// TwinCAT 3 PLC project SPS
// ProgramVersion: 3.1.4024.0
// libraries:
//   Tc2_MC2, * (Beckhoff Automation GmbH)
//   Tc2_Standard, * (Beckhoff Automation GmbH)
//   Tc2_System, * (Beckhoff Automation GmbH)
//   Tc3_IotBase, * (Beckhoff Automation GmbH)
//   Tc3_Module, * (Beckhoff Automation GmbH)
// project tree:
//   DUTs/ eBetriebszustand.TcDUT
//   GVLs/ GVL_PosKinematic.TcGVL, IFC_HW.TcGVL (not stored)
//   / PlcTask.TcTTO
//   POUs/ FB_Abfullmodul.TcPOU, FB_Ampel.TcPOU, FB_Blinklicht.TcPOU, FB_Dispenser.TcPOU, FB_EZylinder.TcPOU, FB_IotMqttCommunication.TcPOU, FB_ManipulatorAchsen.TcPOU, FB_Vereinzelung.TcPOU, FUN_Scale.TcPOU, MAIN.TcPOU
//   POUs/PortalRoboter/ FB_AchsenRoboter.TcPOU, FB_Robotersteuerung.TcPOU, FB_Thermo_Temp.TcPOU, FB_Waage_Temp.TcPOU
//   POUs/Transport/ FB_TransportBand.TcPOU, FB_Transport.TcPOU, FB_TransportA.TcPOU, FB_TransportLogik.TcPOU, FB_TransportE.TcPOU
// real-time tasks:
//   TASK PlcTask: cycle T#10ms, priority 20, ADS port 350
//   TASK PlcTask1: cycle T#10ms, priority 21, ADS port 351
// motion (NC):
//   TASK NC-Task 1 SAF: cycle T#2ms, priority 4, ADS port 501
//   TASK NC-Task 1 SVB: cycle T#10ms, priority 8, ADS port 511
//   AXIS Achse_ManG (id 7)
//     OtherSettings: AllowMotionCmdToSlave=true
//     encoder EncType=1
//       EncPara: ScaleFactorNumerator=0.0025
//         Inc: RefSearchInverse=true, RefSyncInverse=false
//     drive DrvType=5
//       Analog: TorqueSetpointScale=10, ScaleFactorActTorque=0.1
//       TimeComp: TaskDelayCycles=1
//     controller CtrType=1
//       CtrPara: PriorControlFactor=1
//         Observer: BandWidth=20
//   AXIS Achse_Band (id 1)
//     OtherSettings: AllowMotionCmdToSlave=true
//     encoder EncType=1
//     drive DrvType=5
//       Analog: TorqueSetpointScale=10, ScaleFactorActTorque=0.1
//       TimeComp: TaskDelayCycles=1
//     controller CtrType=1
//       CtrPara: PriorControlFactor=1
//         Observer: BandWidth=20
//   AXIS Achse_Dispenser1 (id 2)
//     OtherSettings: AllowMotionCmdToSlave=true
//     encoder EncType=1
//     drive DrvType=5
//       Analog: TorqueSetpointScale=10, ScaleFactorActTorque=0.1
//       TimeComp: TaskDelayCycles=1
//     controller CtrType=1
//       CtrPara: PriorControlFactor=1
//         Observer: BandWidth=20
//   AXIS Achse_Dispenser2 (id 3)
//     OtherSettings: AllowMotionCmdToSlave=true
//     encoder EncType=1
//     drive DrvType=5
//       Analog: TorqueSetpointScale=10, ScaleFactorActTorque=0.1
//       TimeComp: TaskDelayCycles=1
//     controller CtrType=1
//       CtrPara: PriorControlFactor=1
//         Observer: BandWidth=20
//   AXIS Achse_Dispenser3 (id 4)
//     OtherSettings: AllowMotionCmdToSlave=true
//     encoder EncType=1
//     drive DrvType=5
//       Analog: TorqueSetpointScale=10, ScaleFactorActTorque=0.1
//       TimeComp: TaskDelayCycles=1
//     controller CtrType=1
//       CtrPara: PriorControlFactor=1
//         Observer: BandWidth=20
//   AXIS Achse_ManX (id 5)
//     OtherSettings: AllowMotionCmdToSlave=true
//     encoder EncType=1
//       EncPara: ScaleFactorNumerator=0.0025
//         Inc: RefSearchInverse=true, RefSyncInverse=false
//     drive DrvType=5
//       Analog: TorqueSetpointScale=10, ScaleFactorActTorque=0.1
//       TimeComp: TaskDelayCycles=1
//     controller CtrType=1
//       CtrPara: PriorControlFactor=1
//         Observer: BandWidth=20
//   AXIS Achse_ManY (id 6)
//     OtherSettings: AllowMotionCmdToSlave=true
//     encoder EncType=1
//       EncPara: ScaleFactorNumerator=0.0025
//         Inc: RefSearchInverse=true, RefSyncInverse=false
//     drive DrvType=5
//       Analog: TorqueSetpointScale=10, ScaleFactorActTorque=0.1
//       TimeComp: TaskDelayCycles=1
//     controller CtrType=1
//       CtrPara: PriorControlFactor=1
//         Observer: BandWidth=20
//   AXIS Achse_ManZ (id 8)
//     OtherSettings: AllowMotionCmdToSlave=true
//     encoder EncType=1
//       EncPara: ScaleFactorNumerator=0.0025
//         Inc: RefSearchInverse=true, RefSyncInverse=false
//     drive DrvType=5
//       Analog: TorqueSetpointScale=10, ScaleFactorActTorque=0.1
//       TimeComp: TaskDelayCycles=1
//     controller CtrType=1
//       CtrPara: PriorControlFactor=1
//         Observer: BandWidth=20
// I/O:
//   DEVICE Gerät 3 (EtherCAT) (disabled), AmsNetId 192.168.137.1.4.1
//     Klemme 1 (EK1100) [EK1100 EtherCAT-Koppler (2A E-Bus)]
//       Klemme 2 (EL1014) [EL1014 4K. Dig. Eingang 24V, 10µs]
//       Klemme 3 (EL2008) [EL2008 8K. Dig. Ausgang 24V, 0.5A]
//       Klemme 4 (EL2008) [EL2008 8K. Dig. Ausgang 24V, 0.5A]
//       Klemme 5 (EL9011) [EL9011 Endklemme]
// variable links:
//   SPS/SPS Instance <-> Device 3 (EtherCAT)/Term 1 (EK1100)/Term 2 (EL1014)
//     PlcTask Inputs/IFC_HW.bExecute <-> Channel 1/Input
//   SPS/SPS Instance <-> Device 3 (EtherCAT)/Term 1 (EK1100)/Term 3 (EL2008)
//     PlcTask Outputs/IFC_HW.bAmpelRot <-> Channel 1/Output
//   SPS/SPS Instance <-> NC-Task 1 SAF/Axes/Achse_Band
//     PlcTask Inputs/IFC_HW.ax_BandMotor.NcToPlc <-> Outputs/ToPlc
//     PlcTask Outputs/IFC_HW.ax_BandMotor.PlcToNc <-> Inputs/FromPlc
//   SPS/SPS Instance <-> NC-Task 1 SAF/Axes/Achse_Dispenser1
//     PlcTask Inputs/IFC_HW.ax_Extruder1.NcToPlc <-> Outputs/ToPlc
//     PlcTask Outputs/IFC_HW.ax_Extruder1.PlcToNc <-> Inputs/FromPlc
//   SPS/SPS Instance <-> NC-Task 1 SAF/Axes/Achse_Dispenser2
//     PlcTask Inputs/IFC_HW.ax_Extruder2.NcToPlc <-> Outputs/ToPlc
//     PlcTask Outputs/IFC_HW.ax_Extruder2.PlcToNc <-> Inputs/FromPlc
//   SPS/SPS Instance <-> NC-Task 1 SAF/Axes/Achse_Dispenser3
//     PlcTask Inputs/IFC_HW.ax_Extruder3.NcToPlc <-> Outputs/ToPlc
//     PlcTask Outputs/IFC_HW.ax_Extruder3.PlcToNc <-> Inputs/FromPlc
//   SPS/SPS Instance <-> NC-Task 1 SAF/Axes/Achse_ManG
//     PlcTask Inputs/IFC_HW.ax_ManG.NcToPlc <-> Outputs/ToPlc
//     PlcTask Outputs/IFC_HW.ax_ManG.PlcToNc <-> Inputs/FromPlc
//   SPS/SPS Instance <-> NC-Task 1 SAF/Axes/Achse_ManX
//     PlcTask Inputs/IFC_HW.ax_ManX.NcToPlc <-> Outputs/ToPlc
//     PlcTask Outputs/IFC_HW.ax_ManX.PlcToNc <-> Inputs/FromPlc
//   SPS/SPS Instance <-> NC-Task 1 SAF/Axes/Achse_ManY
//     PlcTask Inputs/IFC_HW.ax_ManY.NcToPlc <-> Outputs/ToPlc
//     PlcTask Outputs/IFC_HW.ax_ManY.PlcToNc <-> Inputs/FromPlc
//   SPS/SPS Instance <-> NC-Task 1 SAF/Axes/Achse_ManZ
//     PlcTask Inputs/IFC_HW.ax_ManZ.NcToPlc <-> Outputs/ToPlc
//     PlcTask Outputs/IFC_HW.ax_ManZ.PlcToNc <-> Inputs/FromPlc

CONFIGURATION SPS
    RESOURCE PLC ON TwinCAT3
        TASK PlcTask(INTERVAL := T#10ms, PRIORITY := 20);
        PROGRAM MAIN WITH PlcTask : MAIN;
    END_RESOURCE
END_CONFIGURATION

// ---- DUTs/eBetriebszustand.TcDUT
{attribute 'qualified_only'}
{attribute 'strict'}
TYPE eBetriebszustand :
(
	Off , //Nicht Betriebsbereit, ROT
	Error , //Fehlerbehafteter Stop (Sicherheitssteuerung), ROT blinkend
	Setup , //Wartung, GELB
	Warning , //Nicht Fehlerbehafteter aber nicht geplanter Stop, GELB blinkend
	Init ,  //herstellung Betriebsbereitschaft, GELB GRÜN
	Ready , // Betriebsbereitschaft, GRÜN
	Production , //Betrieb, GRÜN GELB blinkend
	Done, //Betrieb abgeschlossen, GRÜN blinkend
	Stop //Geplanter Stopp ROT GELB blinkend
	
);
END_TYPE

// ---- GVLs/GVL_PosKinematic.TcGVL
{attribute 'qualified_only'}
VAR_GLOBAL
	// Home position
	pXhome : REAL := 29;
	pYhome : REAL := 145.5;
	pZhome : REAL := 45;
	
	// Conveyor position
	pXconv : REAL := 29;
	pYconv : REAL := 145.5;
	pZconv : REAL := 130;
	
	//Scale position
	pXscale : REAL := 36;
	pYscale : REAL := 7.5;
	pZscale : REAL := 131.5;
	
	// Heating position
	pXheat : REAL := 218.5;
	pYheat : REAL := 7;
	pZheat : REAL := 159;
	
	// Storage position
	pX1stor : REAL := 107;
	pX2stor : REAL := 158.7;
	pX3stor : REAL := 209.3;
	pX4stor : REAL := 260.3;
	pYstor : REAL := 139;
	pZstor : REAL := 120;
	
	// Z offset height
	pZoff : REAL := 45;
END_VAR

// ---- POUs/MAIN.TcPOU
PROGRAM MAIN
VAR
	fbAmpel : FB_Ampel;
	fbEZylinder1 : FB_EZylinder;
	fbEZylinder2 : FB_EZylinder;
	MCPowerBand : MC_Power;
	MCPowerDispenser1 	: MC_Power;
	MCPowerDispenser2 	: MC_Power;
	MCPowerDispenser3 	: MC_Power;
	MCPowerAchseX	 	: MC_Power;
	MCPowerAchseY 	: MC_Power;
	MCPowerAchseZ 	: MC_Power;
	MCPowerAchseG 	: MC_Power;
	fbAbfullModul : FB_Abfullmodul;
	fbRoboter : FB_Robotersteuerung;
	fbIotMqttCommunication : FB_IotMqttCommunication;
	
	nRoboterLagerIndex : INT;
	

	ix : REAL;
	ry : UINT;
	
	
  	

END_VAR

ry := TO_UINT(FUN_Scale(ix,4096, 0, 350, 0));

IFC_HW.ax_BandMotor.ReadStatus();
IFC_HW.ax_Extruder1.ReadStatus();
IFC_HW.ax_Extruder2.ReadStatus();
IFC_HW.ax_Extruder3.ReadStatus();



MCPowerBand(
	Axis:= IFC_HW.ax_BandMotor , 
	Enable:= TRUE , 
	Enable_Positive:= TRUE, 
	Enable_Negative:= TRUE, 
	Override:= , 
	BufferMode:= , 
	Options:= , 
	Status=> , 
	Busy=> , 
	Error=> , 
	ErrorID=> );
	
MCPowerDispenser1(
	Axis:= IFC_HW.ax_Extruder1, 
	Enable:= TRUE, 
	Enable_Positive:= TRUE, 
	Enable_Negative:= TRUE, 
	Override:= , 
	BufferMode:= , 
	Options:= , 
	Status=> , 
	Busy=> , 
	Error=> , 
	ErrorID=> );
	
MCPowerDispenser2(
	Axis:= IFC_HW.ax_Extruder2, 
	Enable:= TRUE, 
	Enable_Positive:= TRUE, 
	Enable_Negative:= TRUE, 
	Override:= , 
	BufferMode:= , 
	Options:= , 
	Status=> , 
	Busy=> , 
	Error=> , 
	ErrorID=> );
	
MCPowerDispenser3(
	Axis:= IFC_HW.ax_Extruder3, 
	Enable:= TRUE, 
	Enable_Positive:= TRUE, 
	Enable_Negative:= TRUE, 
	Override:= , 
	BufferMode:= , 
	Options:= , 
	Status=> , 
	Busy=> , 
	Error=> , 
	ErrorID=> );
	
MCPowerAchseX(
	Axis:= IFC_HW.ax_ManX, 
	Enable:= TRUE, 
	Enable_Positive:= TRUE, 
	Enable_Negative:= TRUE, 
	Override:= , 
	BufferMode:= , 
	Options:= , 
	Status=> , 
	Busy=> , 
	Error=> , 
	ErrorID=> );
	
MCPowerAchseY(
	Axis:= IFC_HW.ax_ManY, 
	Enable:= TRUE, 
	Enable_Positive:= TRUE, 
	Enable_Negative:= TRUE, 
	Override:= , 
	BufferMode:= , 
	Options:= , 
	Status=> , 
	Busy=> , 
	Error=> , 
	ErrorID=> );

MCPowerAchseZ(
	Axis:= IFC_HW.ax_ManZ, 
	Enable:= TRUE, 
	Enable_Positive:= TRUE, 
	Enable_Negative:= TRUE, 
	Override:= , 
	BufferMode:= , 
	Options:= , 
	Status=> , 
	Busy=> , 
	Error=> , 
	ErrorID=> );
	
MCPowerAchseG(
	Axis:= IFC_HW.ax_ManG, 
	Enable:= TRUE, 
	Enable_Positive:= TRUE, 
	Enable_Negative:= TRUE, 
	Override:= , 
	BufferMode:= , 
	Options:= , 
	Status=> , 
	Busy=> , 
	Error=> , 
	ErrorID=> );


fbAbfullModul(
	bEnable:= IFC_HW.bEnable, 
	bExecute:= IFC_HW.bExecute, 
	bBandSens1:= IFC_HW.bBandSens1, 
	bBandSens2:= IFC_HW.bBandSens2, 
	bBandSens3:= IFC_HW.bBandSens3, 
	bBandSens4:= IFC_HW.bBandSens4, 
	bEinzelSens1:= IFC_HW.bEinzelSens1 , 
	bEinzelSens2:= IFC_HW.bEinzelSens2, 
	bEinzelSens3:= IFC_HW.bEinzelSens3, 
	nLagerIndex:= , 
	bGate1=> fbEZylinder1.bGate, 
	bGate2=> fbEZylinder2.bGate, 
	bStopper1=> IFC_HW.bBandHub1 , 
	bStopper2=> IFC_HW.bBandHub2, 
	bStopper3=> IFC_HW.bBandHub3, 
	eState=> , 
	axFoerderband:= IFC_HW.ax_BandMotor, 
	axDispenser1:= IFC_HW.ax_Extruder1, 
	axDispenser2:= IFC_HW.ax_Extruder2, 
	axDispenser3:= IFC_HW.ax_Extruder3
 );
 
 fbRoboter(
    bEnable := IFC_HW.bEnable,
    bExecute := IFC_HW.bExecute,

    bSensBand4 := IFC_HW.bBandSens4,
    bSensEndX := IFC_HW.bManEndXmin,
    bSensEndY := IFC_HW.bManEndYmin,
    bSensEndZ := IFC_HW.bManEndZmin,
    bSensEndG := IFC_HW.bManEndGmin,

    eState => ,

    bBrakeZ => IFC_HW.bManBrakeZ,
    bGripperClosed => IFC_HW.bGripperClosed,

    axX := IFC_HW.ax_ManX,
    axY := IFC_HW.ax_ManY,
    axZ := IFC_HW.ax_ManZ,
    axG := IFC_HW.ax_ManG,

    nLagerIndex := nRoboterLagerIndex
);
 
 fbIotMqttCommunication(
	sTopicToPublish:= 'bEnable',
	sMessageToPublish:= BOOL_TO_STRING(IFC_HW.bEnable),
);
	
fbEZylinder1(bGate:= , bError:= ,
			 bR1=> IFC_HW.bR1AKT1, bR2=> IFC_HW.bR2AKT1);
fbEZylinder2(bGate:= , bError:= , 
			bR1=> IFC_HW.bR1AKT2, bR2=> IFC_HW.bR2AKT2 );
			
fbAmpel(eState:= fbAbfullmodul.eState, bAmpelGrun=> IFC_HW.bAmpelGrun, bAmpelRot=> IFC_HW.bAmpelRot , bAmpelGelb=> IFC_HW.bAmpelGelb);

END_PROGRAM

// ---- POUs/FB_Ampel.TcPOU
FUNCTION_BLOCK FB_Ampel
VAR_INPUT
	eState : eBetriebszustand;
END_VAR
VAR_OUTPUT
	bAmpelGrun : BOOL;
	bAmpelRot : BOOL;
	bAmpelGelb : BOOL;
END_VAR
VAR
	fbBlinklicht : FB_Blinklicht;
END_VAR

CASE eState OF
	eBetriebszustand.Off:
		bAmpelGrun := FALSE;
		bAmpelGelb := FALSE;
		bAmpelRot := TRUE;
	
	eBetriebszustand.Error:
		bAmpelGrun := FALSE;
		bAmpelGelb := FALSE;
		fbBlinklicht(bStartStop:= TRUE, tPeriode:= T#1S, bBlink=> bAmpelRot );
	
	eBetriebszustand.Setup:
		bAmpelGrun := FALSE;
		bAmpelGelb := TRUE;
		bAmpelRot := FALSE;
	
	eBetriebszustand.Warning:
		bAmpelGrun := FALSE;
		fbBlinklicht(bStartStop:= TRUE, tPeriode:= T#1S, bBlink=> bAmpelGelb );
		bAmpelRot := FALSE;
		
	eBetriebszustand.Init:
		bAmpelGrun := TRUE;
		bAmpelGelb := TRUE;
		bAmpelRot := FALSE;
	
	eBetriebszustand.Ready:
		bAmpelGrun := TRUE;
		bAmpelGelb := FALSE;
		bAmpelRot := FALSE;
	
	eBetriebszustand.Production:
		bAmpelRot := FALSE;
		fbBlinklicht(bStartStop:= TRUE , tPeriode:= T#1S, bBlink=> bAmpelGrun);
		fbBlinklicht(bStartStop:= TRUE , tPeriode:= T#1S, bBlink=> bAmpelGelb);
	
	eBetriebszustand.Done:
		fbBlinklicht(bStartStop:= TRUE , tPeriode:= T#1S, bBlink=> bAmpelGrun);
		bAmpelGelb := FALSE;
		bAmpelRot := FALSE;
		
	eBetriebszustand.Stop:
		bAmpelGrun := FALSE;
		fbBlinklicht(bStartStop:= TRUE , tPeriode:= T#1S, bBlink=> bAmpelRot);
		fbBlinklicht(bStartStop:= TRUE , tPeriode:= T#1S, bBlink=> bAmpelGelb);
	
	
	
	
	
	
	
END_CASE

END_FUNCTION_BLOCK

// ---- POUs/FB_Blinklicht.TcPOU
FUNCTION_BLOCK FB_Blinklicht
VAR_INPUT
	bStartStop : BOOL;
	tPeriode : TIME := T#1S;
END_VAR
VAR_OUTPUT
	bBlink : BOOL;
END_VAR
VAR
	fbTon : Ton;
	fbRtrig : R_Trig;
	bEinAus : BOOL;
END_VAR


fbRtrig(CLK:= bStartStop, Q=>);
IF fbRtrig.Q THEN
	bEinAus := NOT bEinAus;
END_IF


//fbTon.IN := bBlink AND NOT fbTon.Q;
//fbTon.PT := T#1S;

fbTon(IN:= bEinAus AND NOT fbTon.Q , PT:= tPeriode , Q=>  , ET=> );

IF fbTon.ET <= fbTon.PT/2 THEN
	bBlink := FALSE;
ELSIF fbTon.ET > fbTon.PT/2 THEN
	bBlink := TRUE;
END_IF

END_FUNCTION_BLOCK

// ---- POUs/FB_EZylinder.TcPOU
FUNCTION_BLOCK FB_EZylinder
VAR_INPUT
	bGate : BOOL;
	bError : BOOL;
END_VAR
VAR_OUTPUT
	bR1 : BOOL;
	bR2 : BOOL;
END_VAR
VAR
END_VAR


bR1 := bGate;
bR2 := NOT bGate;

IF bError THEN
	bR1 := FALSE;
	bR2 := FALSE;
END_IF

END_FUNCTION_BLOCK

// ---- POUs/FB_Abfullmodul.TcPOU
FUNCTION_BLOCK FB_AbfullModul
VAR_INPUT
    bEnable     : BOOL;
    bExecute    : BOOL; 
	bBandSens1 	: BOOL;   
    bBandSens2 	: BOOL; 
	bBandSens3 	: BOOL; 
	bBandSens4 	: BOOL; 
 	bEinzelSens1: BOOL;
	bEinzelSens2: BOOL;
	bEinzelSens3: BOOL;
	nLagerIndex : INT;
END_VAR

VAR_OUTPUT
	//Vereinzelungsoutputs
	bGate1 : BOOL;
    bGate2 : BOOL;
	//Transportoutputs
	bStopper1 : BOOL;
    bStopper2 : BOOL;
    bStopper3 : BOOL;
    eState      : eBetriebszustand;
END_VAR

VAR
    fbVereinzelung      : FB_Vereinzelung;
    fbDispenser1         : FB_Dispenser;
	fbDispenser2         : FB_Dispenser;
	fbDispenser3         : FB_Dispenser;
    fbTransport    		: FB_Transport;
	
	fTrigBandSens4 : f_TRIG; 
	bBandSens4Rise  : BOOL;
	
    nState : INT := 0;
	nStation : INT;
	
	
END_VAR

VAR_IN_OUT
    axFoerderband : Axis_Ref;
    axDispenser1    : Axis_Ref;
	axDispenser2    : Axis_Ref;
	axDispenser3    : Axis_Ref;
   // axManipulator : Axis_Ref;
END_VAR

fbVereinzelung(
	bEnable:= bEnable, 
	bExecute:=  , 
	bSensor1:= bEinzelSens1, 
	bSensor2:= bEinzelSens2 , 
	bSensor3:= bEinzelSens3 , 
	bSensor4:= bBandSens1 , 
	bGate1=> bGate1 , 
	bGate2=> bGate2, 
	eState=> );
	
fbTransport(
	bEnable:= bEnable, 
	bExecute:= , 
	nStation:= nStation, 
	bSens1:= bBandSens1, 
	bSens2:= bBandSens2, 
	bSens3:= bBandSens3 , 
	bSens4:= bBandSens4, 
	eState=> , 
	bStopper1=> bStopper1, 
	bStopper2=> bStopper2, 
	bStopper3=> bStopper3, 
	ax:= axFoerderband);
	
fbDispenser1(
	bEnable:= bEnable, 
	bExecute:=, 
	rDistance:= , 
	eState=> , 
	ax:= axDispenser1);
	
fbDispenser2(
	bEnable:= bEnable, 
	bExecute:=, 
	rDistance:= , 
	eState=> , 
	ax:= axDispenser2);
	
fbDispenser3(
	bEnable:= bEnable, 
	bExecute:= , 
	rDistance:= , 
	eState=> , 
	ax:= axDispenser3);
	
	
CASE nState OF
	0: // OFF
	eState := eBetriebszustand.Off;
	fbVereinzelung.bEnable := FALSE;
	fbVereinzelung.bExecute := FALSE;
	fbTransport.bEnable := FALSE;
	fbTransport.bExecute := FALSE;
	fbDispenser1.bEnable := FALSE;
	fbDispenser2.bEnable := FALSE;
	fbDispenser3.bEnable := FALSE;
	fbDispenser1.bExecute := FALSE;
	fbDispenser2.bExecute := FALSE;
	fbDispenser3.bExecute := FALSE;
	
	
	IF bEnable THEN
		nState := 10;
	END_IF
	
	10: // INIT
	
	eState := eBetriebszustand.Init;
	fbVereinzelung.bEnable := TRUE;
	fbVereinzelung.bExecute := FALSE;
	fbTransport.bEnable := TRUE;
	fbTransport.bExecute := FALSE;
	fbDispenser1.bEnable := TRUE;
	fbDispenser2.bEnable := TRUE;
	fbDispenser3.bEnable := TRUE;
	fbDispenser1.bExecute := FALSE;
	fbDispenser2.bExecute := FALSE;
	fbDispenser3.bExecute := FALSE;
	
	IF fbVereinzelung.eState = eBetriebszustand.Ready AND fbTransport.eState = eBetriebszustand.Ready AND fbDispenser1.eState = eBetriebszustand.Ready AND fbDispenser2.eState = eBetriebszustand.Ready AND fbDispenser3.eState = eBetriebszustand.Ready THEN
		nState := 20;
	END_IF
	
	20: // READY
	eState := eBetriebszustand.Ready;
	fbVereinzelung.bEnable := TRUE;
	fbVereinzelung.bExecute := FALSE;
	fbTransport.bEnable := TRUE;
	fbTransport.bExecute := FALSE;
	fbDispenser1.bEnable := TRUE;
	fbDispenser2.bEnable := TRUE;
	fbDispenser3.bEnable := TRUE;
	fbDispenser1.bExecute := FALSE;
	fbDispenser2.bExecute := FALSE;
	fbDispenser3.bExecute := FALSE;
	
	IF bExecute THEN
		nState := 30;
	END_IF
	
	30: //Production
	eState := eBetriebszustand.Production;
	fbVereinzelung.bExecute := TRUE;
	fbTransport.bExecute := TRUE;
	fbDispenser1.bExecute := FALSE;
	fbDispenser2.bExecute := FALSE;
	fbDispenser3.bExecute := FALSE;
	nStation := 1;
	
	IF fbVereinzelung.eState = eBetriebszustand.Done AND fbTransport.eState = eBetriebszustand.Done THEN
		nState := 31;
	END_IF
	
	31: // 1st Dispenser
	nStation := 1;
	fbDispenser1.bExecute := TRUE;
	fbVereinzelung.bExecute := FALSE;
	fbTransport.bExecute := FALSE;
	
	IF fbDispenser1.eState = eBetriebszustand.Done THEN
		nState := 32;
	END_IF
	
	32: // Bewegung zu Station 2
	nStation := 2;
	fbTransport.bExecute := TRUE;
	fbDispenser1.bExecute := FALSE;
	
	IF fbTransport.eState = eBetriebszustand.Done THEN
		nState := 33;
	END_IF
	
	33: // 2nd Dispenser
	
	fbDispenser2.bExecute := TRUE;
	fbTransport.bExecute := FALSE;
	
	IF fbDispenser2.eState = eBetriebszustand.Done THEN
		nState := 34;
	END_IF
	
	34: //Bewegung zu Station 3
	nStation := 3;
	fbTransport.bExecute := TRUE;
	fbDispenser2.bExecute := FALSE;
	
	IF fbTransport.eState = eBetriebszustand.Done THEN
		nState := 35;
	END_IF
	
	35: //3rd Dispenser
	fbTransport.bExecute := FALSE;
	fbDispenser3.bExecute := TRUE;
	
	IF fbDispenser3.eState = eBetriebszustand.Done THEN
		nState := 36;
	END_IF
	
	36: // Bewegung zu Abholstation
	nStation := 4;
	fbDispenser3.bExecute := FALSE;
	fbTransport.bExecute := TRUE;
	
	IF fbTransport.eState = eBetriebszustand.Done THEN
		nState := 40;
	END_IF
	
	40: //DONE
	eState := eBetriebszustand.Done;
	fbTransport.bExecute := FALSE;
	
	
	IF NOT bExecute THEN
		nState := 20;
	END_IF
	
	
END_CASE

END_FUNCTION_BLOCK

// ---- POUs/FB_Vereinzelung.TcPOU
FUNCTION_BLOCK FB_Vereinzelung
VAR_INPUT
	//Steuervariablen
	bEnable : BOOL;
	bExecute : BOOL;
	//Hardware Eingänge
	bSensor1 : BOOL; // Flasche in der Kammer
	bSensor2 : BOOL; //Flasche im Rohr
	bSensor3 : BOOL; //Flasche auf Kopf
	bSensor4 : BOOL; //Flasche am Förderband
END_VAR
VAR_OUTPUT
	//Hardware Ausgänge
	bGate1 : BOOL;
	bGate2 : BOOL;
	//Steuervariable
	eState : eBetriebszustand;
END_VAR
VAR
	nState : INT := 100;
	fbTon : Ton;
END_VAR

fbTon(IN :=, PT := T#1S, Q=>, ET=>);
CASE nState OF
	100:
	eState := eBetriebszustand.Off;
	
	IF bSensor1 AND bEnable THEN
		nState := 21; //Ready
		ELSIF bEnable THEN
			nState := 0; //Init
	END_IF
	
	0: //Kammer ist Leer
	eState := eBetriebszustand.Init;
	bGate1 := FALSE;
	bGate2 := FALSE;
	
	IF bSensor2 THEN
		nState := 1; //Oben öffnen
	END_IF
	
	1: //Oben öffnen
	eState := eBetriebszustand.Init;
	bGate1 := TRUE;
	bGate2 := FALSE;
	
	IF bSensor1 THEN
		nState := 2; //oben schließen
	END_IF
	
	2: //oben Schließen
	eState := eBetriebszustand.Init;
	bGate1 := FALSE;
	bGate2 := FALSE;
	fbTon.IN := TRUE;
	
	
	IF fbTon.Q THEN
		nState := 21; //Ready
		fbTon.IN := FALSE;

	END_IF
	21: //Ready
	eState := eBetriebszustand.Ready;
	bGate1 := FALSE;
	bGate2 := FALSE;
	
	IF bExecute THEN
		nState := 3;
	END_IF
	
	3:
	eState := eBetriebszustand.Production;
	bGate1 := FALSE;
	bGate2 := TRUE;
	
	IF bSensor4 THEN
		nState := 4;
	END_IF
	
	4:
	eState := eBetriebszustand.Production;
	bGate1 := FALSE;
	bGate2 := FALSE;
	fbTon.IN := TRUE;
	
	IF fbTon.Q THEN
		nState := 41;
		fbTon.IN := FALSE;
		
	END_IF
	
	41: 
	eState := eBetriebszustand.Done;
	
	IF NOT bExecute THEN
		nState := 0;
		
	END_IF
	
	IF NOT bSensor2 AND bSensor3 THEN
		nState := 33;
	END_IF
	
	33:
	eState := eBetriebszustand.Warning;
	
	bExecute := FALSE;
	
	

	
END_CASE

END_FUNCTION_BLOCK

// ---- POUs/FB_Dispenser.TcPOU
FUNCTION_BLOCK FB_Dispenser
VAR_INPUT
	bEnable : BOOL;
	bExecute : BOOL;
	rDistance : REAL;
	
END_VAR
VAR_OUTPUT
	eState : eBetriebszustand;
END_VAR
VAR
	mcReset : MC_Reset;
	mcPower : MC_Power;
	mcMoveRelative : MC_MoveRelative;
	nState : INT;
END_VAR

VAR_IN_OUT
	// Achsen Ref
	ax : Axis_Ref;
END_VAR

ax.ReadStatus();

mcReset(
	Axis:= ax, 
	Execute:= , 
	Done=> , 
	Busy=> , 
	Error=> , 
	ErrorID=> );

mcPower(
	Axis:= ax, 
	Enable:= , 
	Enable_Positive:= , 
	Enable_Negative:= , 
	Override:= , 
	BufferMode:= , 
	Options:= , 
	Status=> , 
	Busy=> , 
	Error=> , 
	ErrorID=> );
	
mcMoveRelative(
	Axis:= ax, 
	Execute:= , 
	Distance:= 10, 
	Velocity:= , 
	Acceleration:= , 
	Deceleration:= , 
	Jerk:= , 
	BufferMode:= , 
	Options:= , 
	Done=> , 
	Busy=> , 
	Active=> , 
	CommandAborted=> , 
	Error=> , 
	ErrorID=> );
	
IF NOT mcPower.Status THEN
	nState := 0;
END_IF

CASE nState OF
	0: // OFF
	eState := eBetriebszustand.Off;
	mcPower.Enable := TRUE;
	mcPower.Enable_Positive := TRUE;
	IF bEnable AND mcPower.Status THEN
		nState := 20; //Ready
	ELSIF bEnable AND NOT mcPower.Status THEN
		nState := 10; // Init-Rest
	END_IF
	
	
	10: // Init - Reset
	eState := eBetriebszustand.Init;
	mcReset.Execute := TRUE;
	mcPower.Enable := FALSE;
	IF mcReset.Done THEN
		mcReset.Execute := FALSE;
		nState := 11;
	END_IF
	
	11: // Init - Power
	eState := eBetriebszustand.Init;
	mcPower.Enable := TRUE;
	mcReset.Execute := FALSE;
	IF mcPower.Status THEN
		nState := 20;
	END_IF
	
	20: //Ready
	eState := eBetriebszustand.Ready;
	IF bExecute THEN
		nState := 30;
	END_IF
	
	30: //Production
	eState := eBetriebszustand.Production;
	mcMoveRelative.Execute := TRUE;
	mcMoveRelative.Velocity := 20;
	mcMoveRelative.Acceleration := 20;
	mcMoveRelative.Distance := rDistance;
	
	IF mcMoveRelative.Done THEN
		nState := 40;
	END_IF
	
	40: // Fertig
	eState := eBetriebszustand.Done;
	mcMoveRelative.Execute := FALSE;
	
	IF NOT bExecute THEN
		nState := 20;
	END_IF
END_CASE

END_FUNCTION_BLOCK

// ---- POUs/Transport/FB_Transport.TcPOU
FUNCTION_BLOCK FB_Transport
VAR_INPUT
	bEnable : BOOL;
	bExecute : BOOL;
	nStation : INT;
	//Hardware Eingänge
	bSens1 : BOOL;
	bSens2 : BOOL;
	bSens3 : BOOL;
	bSens4 : BOOL;
	
END_VAR
VAR_OUTPUT
	eState : eBetriebszustand;
	bStopper1 : BOOL;
	bStopper2 : BOOL;
	bStopper3 : BOOL;
END_VAR
VAR
	fbTransportE : FB_TransportE;
	fbTransportLogik : FB_TransportLogik;
	fbTransportBand : FB_TransportBand;
	fbTransportA : FB_TransportA;
	
	
END_VAR
VAR_IN_OUT
	// Achsen Ref
	ax : Axis_Ref;
END_VAR

fbTransportE(
	bSens1:= bSens1, 
	bSens2:= bSens2, 
	bSens3:= bSens3 , 
	bSens4:= bSens4, 
	bStation1=> , 
	bStation2=> , 
	bStation3=> , 
	bStation4=> );
	
fbTransportLogik(
	bEnable:= bEnable, 
	bExecute:= bExecute , 
	eStateE:= fbTransportBand.eState , 
	nStation:= nStation, 
	bStation1:= fbTransportE.bStation1, 
	bStation2:= fbTransportE.bStation2, 
	bStation3:= fbTransportE.bStation3, 
	bStation4:= fbTransportE.bStation4, 
	bEnableA=> , 
	bExecuteA=> , 
	bStopA=> , 
	eStateA=> eState, 
	bStop1=> , 
	bStop2=> , 
	bStop3=> );
	
fbTransportBand(
	bEnable:= fbTransportLogik.bEnableA , 
	bExecute:= fbTransportLogik.bExecuteA, 
	bHalt:= fbTransportLogik.bStopA, 
	eState=>, 
	ax:= ax);
	
fbTransportA(
	bStop1:= fbTransportLogik.bStop1 , 
	bStop2:= fbTransportLogik.bStop2, 
	bStop3:= fbTransportLogik.bStop3, 
	bStopper1=> bStopper1, 
	bStopper2=> bStopper2, 
	bStopper3=> bStopper3);

END_FUNCTION_BLOCK

// ---- POUs/Transport/FB_TransportE.TcPOU
FUNCTION_BLOCK FB_TransportE
VAR_INPUT
	//Hardware Signale
	bSens1 : BOOL;
	bSens2 : BOOL;
	bSens3 : BOOL;
	bSens4 : BOOL;
	
END_VAR
VAR_OUTPUT
	bStation1 : BOOL;
	bStation2 : BOOL;
	bStation3 : BOOL;
	bStation4 : BOOL;
END_VAR
VAR
END_VAR

bStation1 := bSens1;
bStation2 := bSens2;
bStation3 := bSens3;
bStation4 := bSens4;

END_FUNCTION_BLOCK

// ---- POUs/Transport/FB_TransportLogik.TcPOU
FUNCTION_BLOCK FB_TransportLogik
VAR_INPUT
	bEnable : BOOL;
	bExecute : BOOL;
	eStateE : eBetriebszustand;
	nStation : INT;
	// Logik -> Hardware Signal
	bStation1 : BOOL;
	bStation2 : BOOL;
	bStation3 : BOOL;
	bStation4 : BOOL; 
END_VAR
VAR_OUTPUT
	bEnableA : BOOL;
	bExecuteA : BOOL;
	bStopA : BOOL;
	eStateA : eBetriebszustand;
	// Hardware Signale -> Logik
	bStop1 : BOOL;
	bStop2 : BOOL;
	bStop3 : BOOL;
	
 
END_VAR
VAR
	nState : INT;
END_VAR

CASE nState OF
	0: // OFF
	bEnableA := FALSE;
	bExecuteA := FALSE;
	bStopA := FALSE;
	eStateA := eBetriebszustand.Off;
	
	IF bEnable THEN
		nState := 1;
	END_IF
	
	1: //INIT
	bEnableA := TRUE;
	bExecuteA := FALSE;
	bStopA := FALSE;
	eStateA := eBetriebszustand.Init;
	
	IF eStateE = eBetriebszustand.Ready THEN
		nState := 2; // Ready
	END_IF
	
	2: // READY
	bEnableA := TRUE;
	bExecuteA := FALSE;
	bStopA := FALSE;
	eStateA := eBetriebszustand.Ready;
	
	IF bExecute THEN
		nState := 3;
	END_IF
	
	3: // FB TransportBand start
	bExecuteA := TRUE;
	eStateA := eBetriebszustand.Production;
	
	IF (nStation - 1) = 1 THEN
		bStop1 := TRUE;
	ELSIF (nStation - 1) = 2 THEN
		bStop2 :=TRUE;
	ELSIF (nStation - 1) = 3 THEN
		bStop3 := TRUE;
	END_IF
	
	IF bStation1 AND (nStation = 1) THEN
		nState := 4;
	ELSIF bStation2 AND (nStation = 2) THEN
		nState := 4;
	ELSIF bStation3 AND (nStation = 3) THEN
		nState := 4;
	ELSIF bStation4 AND (nStation = 4) THEN
		nState := 4;
	END_IF
	
	4: // TransportBand Stop
	
	bExecuteA := FALSE;
	bStopA := TRUE;
	eStateA := eBetriebszustand.Production;
	
	IF (nStation - 1) = 1 THEN
		bStop1 := FALSE;
	ELSIF (nStation - 1) = 2 THEN
		bStop2 := FALSE;
	ELSIF (nStation - 1) = 3 THEN
		bStop3 := FALSE;
	END_IF
	
	IF eStateE = eBetriebszustand.Done THEN
		nState := 5;
	END_IF
	
	5: // DONE
	eStateA := eBetriebszustand.Done;
	
	IF NOT bExecute THEN
		nState := 2;
	END_IF
	
	
	
	
END_CASE

END_FUNCTION_BLOCK

// ---- POUs/Transport/FB_TransportBand.TcPOU
FUNCTION_BLOCK FB_TransportBand
VAR_INPUT
	bEnable : BOOL;
	bExecute : BOOL;
	bHalt : BOOL;
END_VAR

VAR_OUTPUT
	eState : eBetriebszustand;
END_VAR
VAR
	nState : INT := 0;
	rVelocity : REAL;
	rAcceleration : REAL;
	bHaltStart : BOOL := FALSE; // Hilfsvariable, um Halt-Vorgang zu steuern
	// Motionblöcke der Tc2_Mc2
	mcReset : MC_Reset;
	mcPower : MC_Power;
	mcVelocity : MC_MoveVelocity;
	mcHalt : MC_Halt;
END_VAR

VAR_IN_OUT
	ax : Axis_Ref;
END_VAR

ax.ReadStatus();
mcReset(
	Axis:= ax, 
	Execute:= , 
	Done=> , 
	Busy=> , 
	Error=> , 
	ErrorID=> );
	
mcPower(
	Axis:= ax, 
	Enable:= , 
	Enable_Positive:= , 
	Enable_Negative:= , 
	Override:= , 
	BufferMode:= , 
	Options:= , 
	Status=> , 
	Busy=> , 
	Error=> , 
	ErrorID=> );

mcVelocity(
	Axis:= ax, 
	Execute:= , 
	Velocity:= 30, 
	Acceleration:= 60, 
	Deceleration:= , 
	Jerk:= , 
	Direction:= MC_Positive_Direction, 
	BufferMode:= , 
	Options:= , 
	InVelocity=> , 
	Busy=> , 
	Active=> , 
	CommandAborted=> , 
	Error=> , 
	ErrorID=> );
	
mcHalt(
	Axis:= ax, 
	Execute:= , 
	Deceleration:= 10, 
	Jerk:= , 
	BufferMode:= , 
	Options:= , 
	Done=> , 
	Busy=> , 
	Active=> , 
	CommandAborted=> , 
	Error=> , 
	ErrorID=> );

	

IF NOT mcPower.Status THEN
	nState := 0;
END_IF

CASE nState OF
	0: //OFF
	eState := eBetriebszustand.Off;
	mcPower.Enable := TRUE;
	mcPower.Enable_Positive := TRUE;
	// Fehler in der Init Logik
	IF bEnable AND mcPower.Status THEN
		nState := 20; // Ready
	ELSIF bEnable AND NOT mcPower.Status THEN
		nState := 10; // Init-Rest
	END_IF
	
	10: //Init - Reset
	eState := eBetriebszustand.Init;
	mcReset.Execute := TRUE;
	mcPower.Enable := FALSE;
	IF mcReset.Done THEN
		mcReset.Execute := FALSE;
		nState := 11;
	END_IF
	
	11: // Init - Power
	eState := eBetriebszustand.Init;
	mcPower.Enable := TRUE;
	mcReset.Execute := FALSE;
	IF mcPower.Status THEN
		nState := 20;
	END_IF
	
	20: //Ready
	eState := eBetriebszustand.Ready;
	IF bExecute THEN
		nState := 30;
	END_IF
	
	30: //Production
	eState := eBetriebszustand.Production;
	mcVelocity.Execute := TRUE;
	mcVelocity.Velocity := rVelocity;
	mcVelocity.Acceleration := rAcceleration;
	mcVelocity.Direction := MC_Positive_Direction;
	
	IF bHalt THEN 
		mcVelocity.Execute := FALSE;
		nState := 31;
	END_IF
	
	31: // Halten
	eState := eBetriebszustand.Production;
	mcHalt.Execute := TRUE;
	
	IF mcHalt.Done THEN
		nState := 40;
	END_IF
	
	
	40: // Fertig
	eState := eBetriebszustand.Done;
	mcHalt.Execute := FALSE;
	
	IF NOT bExecute THEN
		nState := 20; 
	END_IF
END_CASE

END_FUNCTION_BLOCK

// ---- POUs/Transport/FB_TransportA.TcPOU
FUNCTION_BLOCK FB_TransportA
VAR_INPUT
	bStop1: BOOL;
	bStop2: BOOL;
	bStop3: BOOL;
	
END_VAR
VAR_OUTPUT
	// Hardware Signale
	bStopper1 : BOOL;
	bStopper2 : BOOL;
	bStopper3 : BOOL;
	
END_VAR
VAR
END_VAR

bStopper1 := bStop1;
bStopper2 := bStop2;
bStopper3 := bStop3;

END_FUNCTION_BLOCK

// ---- POUs/PortalRoboter/FB_Robotersteuerung.TcPOU
FUNCTION_BLOCK FB_Robotersteuerung
VAR_INPUT
    bEnable     : BOOL;
    bExecute    : BOOL;

	bSensBand4 	: BOOL;
	bSensEndX : BOOL;		// Manipulator min Endschalter Achse x
	bSensEndY : BOOL;		// Manipulator min Endschalter Achse y
	bSensEndZ : BOOL;		// Manipulator min Endschalter Achse z
	bSensEndG : BOOL;		// Manipulator min Endschalter Achse Gripper
END_VAR

VAR_OUTPUT
    eState          : eBetriebszustand;
    bBrakeZ         : BOOL;
    bGripperClosed  : BOOL;
END_VAR

VAR_IN_OUT
    axX : Axis_Ref;
    axY : Axis_Ref;
    axZ : Axis_Ref;
	axG : Axis_Ref;
	
	nLagerIndex : INT; 
END_VAR

VAR
    fbAchseX : FB_AchsenRoboter;
    fbAchseY : FB_AchsenRoboter;
    fbAchseZ : FB_AchsenRoboter;
	fbAchseG : FB_AchsenRoboter;
	
    fbWaage : FB_Waage_Temp;
    fbThermo : FB_Thermo_Temp;
	
	bCmdX, bCmdY, bCmdZ, bCmdG : BOOL;


	
    bGreifer : BOOL;
    nState   : INT;
END_VAR

// Axis FB calls (using your new sensor variable names)
fbAchseX(
    bEnable := bEnable,
    bExecute := , // filled in per state
    rPosition := ,
    bSensEndstop := bSensEndX,
    eState => ,
    ax := axX);

fbAchseY(
    bEnable := bEnable,
    bExecute := ,
    rPosition := ,
    bSensEndstop := bSensEndY,
    eState => ,
    ax := axY);

fbAchseZ(
    bEnable := bEnable,
    bExecute := ,
    rPosition := ,
    bSensEndstop := bSensEndZ,
    eState => ,
    ax := axZ);

fbAchseG(
    bEnable := bEnable,
    bExecute := ,
    rPosition := ,
    bSensEndstop := bSensEndG,
    eState => ,
    ax := axG);

fbWaage();
fbThermo();

CASE nState OF

0:
    eState := eBetriebszustand.Off;
    bBrakeZ := FALSE;
    bGripperClosed := FALSE;
    nLagerIndex := 1;

    fbAchseG(bExecute := TRUE, rPosition := 7.0, ax := axG);

    IF bEnable THEN
        nState := 10;
    END_IF

10:
    eState := eBetriebszustand.Init;
    bBrakeZ := FALSE;

    fbAchseX(bExecute := TRUE, rPosition := GVL_PosKinematic.pXhome, ax := axX);
    fbAchseY(bExecute := TRUE, rPosition := GVL_PosKinematic.pYhome, ax := axY);
    fbAchseZ(bExecute := TRUE, rPosition := GVL_PosKinematic.pZhome, ax := axZ);

    IF fbAchseX.eState = eBetriebszustand.Done AND
       fbAchseY.eState = eBetriebszustand.Done AND
       fbAchseZ.eState = eBetriebszustand.Done THEN
        fbAchseX.bExecute := FALSE;
        fbAchseY.bExecute := FALSE;
        fbAchseZ.bExecute := FALSE;
        nState := 20;
    END_IF

20:
    eState := eBetriebszustand.Ready;

    IF bSensBand4 THEN
        nState := 30;
    END_IF

30:
    bBrakeZ := TRUE;
    fbAchseZ(bExecute := TRUE, rPosition := GVL_PosKinematic.pZoff, ax := axZ);

    IF fbAchseZ.eState = eBetriebszustand.Done THEN
        fbAchseZ.bExecute := FALSE;
        nState := 31;
    END_IF

31:
    IF fbAchseZ.rPosition <= GVL_PosKinematic.pZoff THEN
        bBrakeZ := FALSE;
        fbAchseX(bExecute := TRUE, rPosition := GVL_PosKinematic.pXconv, ax := axX);
        fbAchseY(bExecute := TRUE, rPosition := GVL_PosKinematic.pYconv, ax := axY);
        IF fbAchseX.eState = eBetriebszustand.Done AND
           fbAchseY.eState = eBetriebszustand.Done THEN
            fbAchseX.bExecute := FALSE;
            fbAchseY.bExecute := FALSE;
            nState := 32;
        END_IF
    END_IF

32:
    IF fbAchseX.rPosition = GVL_PosKinematic.pXconv AND
       fbAchseY.rPosition = GVL_PosKinematic.pYconv THEN
        bBrakeZ := TRUE;
        fbAchseZ(bExecute := TRUE, rPosition := GVL_PosKinematic.pZconv, ax := axZ);
        IF fbAchseZ.eState = eBetriebszustand.Done THEN
            fbAchseZ.bExecute := FALSE;
            nState := 33;
        END_IF
    END_IF

33:
    IF fbAchseZ.rPosition = GVL_PosKinematic.pZconv THEN
        bBrakeZ := FALSE;
        fbAchseG(bExecute := TRUE, rPosition := 9.4, ax := axG);
        IF fbAchseG.eState = eBetriebszustand.Done THEN
            fbAchseG.bExecute := FALSE;
            bGripperClosed := TRUE;
            nState := 34;
        END_IF
    END_IF

34:
    IF fbAchseG.rPosition = 9.4 THEN
        bBrakeZ := TRUE;
        fbAchseZ(bExecute := TRUE, rPosition := GVL_PosKinematic.pZoff, ax := axZ);
        IF fbAchseZ.eState = eBetriebszustand.Done THEN
            fbAchseZ.bExecute := FALSE;
            nState := 40;
        END_IF
    END_IF

40:
    IF fbAchseZ.rPosition <= GVL_PosKinematic.pZoff THEN
        bBrakeZ := FALSE;
        fbAchseX(bExecute := TRUE, rPosition := GVL_PosKinematic.pXscale, ax := axX);
        fbAchseY(bExecute := TRUE, rPosition := GVL_PosKinematic.pYscale, ax := axY);
        IF fbAchseX.eState = eBetriebszustand.Done AND
           fbAchseY.eState = eBetriebszustand.Done THEN
            fbAchseX.bExecute := FALSE;
            fbAchseY.bExecute := FALSE;
            nState := 41;
        END_IF
    END_IF

41:
    IF fbAchseX.rPosition = GVL_PosKinematic.pXscale AND
       fbAchseY.rPosition = GVL_PosKinematic.pYscale THEN
        bBrakeZ := TRUE;
        fbAchseZ(bExecute := TRUE, rPosition := GVL_PosKinematic.pZscale, ax := axZ);
        IF fbAchseZ.eState = eBetriebszustand.Done THEN
            fbAchseZ.bExecute := FALSE;
            nState := 42;
        END_IF
    END_IF

42:
    IF fbAchseZ.rPosition = GVL_PosKinematic.pZscale THEN
        bBrakeZ := FALSE;
        fbAchseG(bExecute := TRUE, rPosition := 7.0, ax := axG);
        IF fbAchseG.eState = eBetriebszustand.Done THEN
            fbAchseG.bExecute := FALSE;
            bGripperClosed := FALSE;
            nState := 43;
        END_IF
    END_IF

43:
    fbWaage(bEnable := TRUE, bExecute := TRUE);
    IF fbWaage.eState = eBetriebszustand.Done THEN
        fbWaage.bExecute := FALSE;
        nState := 44;
    END_IF

44:
    IF NOT fbWaage.bExecute THEN
        fbAchseG(bExecute := TRUE, rPosition := 9.4, ax := axG);
        IF fbAchseG.eState = eBetriebszustand.Done THEN
            fbAchseG.bExecute := FALSE;
            bGripperClosed := TRUE;
            nState := 45;
        END_IF
    END_IF

45:
    IF fbAchseG.rPosition = 9.4 THEN
        bBrakeZ := TRUE;
        fbAchseZ(bExecute := TRUE, rPosition := GVL_PosKinematic.pZoff, ax := axZ);
        IF fbAchseZ.eState = eBetriebszustand.Done THEN
            fbAchseZ.bExecute := FALSE;
            nState := 50;
        END_IF
    END_IF

50:
    IF fbAchseZ.rPosition <= GVL_PosKinematic.pZoff THEN
        bBrakeZ := FALSE;
        fbAchseX(bExecute := TRUE, rPosition := GVL_PosKinematic.pXheat, ax := axX);
        fbAchseY(bExecute := TRUE, rPosition := GVL_PosKinematic.pYheat, ax := axY);
        IF fbAchseX.eState = eBetriebszustand.Done AND
           fbAchseY.eState = eBetriebszustand.Done THEN
            fbAchseX.bExecute := FALSE;
            fbAchseY.bExecute := FALSE;
            nState := 51;
        END_IF
    END_IF

51:
    IF fbAchseX.rPosition = GVL_PosKinematic.pXheat AND
       fbAchseY.rPosition = GVL_PosKinematic.pYheat THEN
        bBrakeZ := TRUE;
        fbAchseZ(bExecute := TRUE, rPosition := GVL_PosKinematic.pZheat, ax := axZ);
        IF fbAchseZ.eState = eBetriebszustand.Done THEN
            fbAchseZ.bExecute := FALSE;
            nState := 52;
        END_IF
    END_IF

52:
    IF fbAchseZ.rPosition = GVL_PosKinematic.pZheat THEN
        bBrakeZ := FALSE;
        fbAchseG(bExecute := TRUE, rPosition := 7.0, ax := axG);
        IF fbAchseG.eState = eBetriebszustand.Done THEN
            fbAchseG.bExecute := FALSE;
            bGripperClosed := FALSE;
            nState := 53;
        END_IF
    END_IF

53:
    fbThermo(bEnable := TRUE, bExecute := TRUE);
    IF fbThermo.eState = eBetriebszustand.Done THEN
        fbThermo.bExecute := FALSE;
        nState := 54;
    END_IF

54:
    IF NOT fbThermo.bExecute THEN
        fbAchseG(bExecute := TRUE, rPosition := 9.4, ax := axG);
        IF fbAchseG.eState = eBetriebszustand.Done THEN
            fbAchseG.bExecute := FALSE;
            bGripperClosed := TRUE;
            nState := 55;
        END_IF
    END_IF

55:
    IF fbAchseG.rPosition = 9.4 THEN
        bBrakeZ := TRUE;
        fbAchseZ(bExecute := TRUE, rPosition := GVL_PosKinematic.pZoff, ax := axZ);
        IF fbAchseZ.eState = eBetriebszustand.Done THEN
            fbAchseZ.bExecute := FALSE;
            bBrakeZ := FALSE;
            nState := 60;
        END_IF
    END_IF

60:
    IF fbAchseZ.rPosition <= GVL_PosKinematic.pZoff THEN
        CASE nLagerIndex OF
            1: fbAchseX.rPosition := GVL_PosKinematic.pX1stor;
            2: fbAchseX.rPosition := GVL_PosKinematic.pX2stor;
            3: fbAchseX.rPosition := GVL_PosKinematic.pX3stor;
            4: fbAchseX.rPosition := GVL_PosKinematic.pX4stor;
            ELSE fbAchseX.rPosition := GVL_PosKinematic.pX1stor;
        END_CASE

        fbAchseX(bExecute := TRUE, ax := axX);
        fbAchseY(bExecute := TRUE, rPosition := GVL_PosKinematic.pYstor, ax := axY);

        IF fbAchseX.eState = eBetriebszustand.Done AND
           fbAchseY.eState = eBetriebszustand.Done THEN
            fbAchseX.bExecute := FALSE;
            fbAchseY.bExecute := FALSE;
            nState := 61;
        END_IF
    END_IF

61:
    IF fbAchseY.rPosition = GVL_PosKinematic.pYstor THEN
        bBrakeZ := TRUE;
        fbAchseZ(bExecute := TRUE, rPosition := GVL_PosKinematic.pZstor, ax := axZ);
        IF fbAchseZ.eState = eBetriebszustand.Done THEN
            fbAchseZ.bExecute := FALSE;
            nState := 62;
        END_IF
    END_IF

62:
    IF fbAchseZ.rPosition = GVL_PosKinematic.pZstor THEN
        bBrakeZ := FALSE;
        fbAchseG(bExecute := TRUE, rPosition := 7.0, ax := axG);
        IF fbAchseG.eState = eBetriebszustand.Done THEN
            fbAchseG.bExecute := FALSE;
            bGripperClosed := FALSE;
            nState := 70;
        END_IF
    END_IF

70:
    IF fbAchseG.rPosition = 7.0 THEN
        bBrakeZ := TRUE;
        fbAchseZ(bExecute := TRUE, rPosition := GVL_PosKinematic.pZoff, ax := axZ);
        IF fbAchseZ.eState = eBetriebszustand.Done THEN
            fbAchseZ.bExecute := FALSE;
            nState := 71;
        END_IF
    END_IF

71:
    IF fbAchseZ.rPosition <= GVL_PosKinematic.pZoff THEN
        bBrakeZ := FALSE;
        fbAchseX(bExecute := TRUE, rPosition := GVL_PosKinematic.pXhome, ax := axX);
        fbAchseY(bExecute := TRUE, rPosition := GVL_PosKinematic.pYhome, ax := axY);
        IF fbAchseX.eState = eBetriebszustand.Done AND
           fbAchseY.eState = eBetriebszustand.Done THEN
            fbAchseX.bExecute := FALSE;
            fbAchseY.bExecute := FALSE;
            nState := 72;
        END_IF
    END_IF

72:
    IF fbAchseX.rPosition = GVL_PosKinematic.pXhome AND
       fbAchseY.rPosition = GVL_PosKinematic.pYhome THEN
        bBrakeZ := TRUE;
        fbAchseZ(bExecute := TRUE, rPosition := GVL_PosKinematic.pZhome, ax := axZ);
        IF fbAchseZ.eState = eBetriebszustand.Done THEN
            fbAchseZ.bExecute := FALSE;
            nState := 80;
        END_IF
    END_IF

80:
    eState := eBetriebszustand.Done;
    bBrakeZ := FALSE;

    IF nLagerIndex < 4 THEN
        nLagerIndex := nLagerIndex + 1;
    ELSE
        nLagerIndex := 1;
    END_IF

    IF NOT bExecute THEN
        nState := 20;
    END_IF

END_CASE

END_FUNCTION_BLOCK

// ---- POUs/PortalRoboter/FB_AchsenRoboter.TcPOU
FUNCTION_BLOCK FB_AchsenRoboter
VAR_INPUT
	bEnable        	: BOOL;
    bExecute       	: BOOL;
    rPosition      	: REAL;
    bSensEndstop    : BOOL;
	bMoveing    	: BOOL;
END_VAR
VAR_OUTPUT
	eState			: eBetriebszustand;
END_VAR
VAR_IN_OUT
	ax				: Axis_Ref;
END_VAR
VAR
	mcPower     	: MC_Power;
    mcMoveAbs   	: MC_MoveAbsolute;
    mcHome      	: MC_Home;
	mcReset			: MC_Reset;
	
	bExecuteLast 	: BOOL;
    bHomeingDone     : BOOL;
    nState      	: INT := 0;
END_VAR

ax.ReadStatus();

mcReset(
	Axis:= ax, 
	Execute:= , 
	Done=> , 
	Busy=> , 
	Error=> , 
	ErrorID=> );

mcPower(
	Axis:= ax, 
	Enable:= , 
	Enable_Positive:= , 
	Enable_Negative:= , 
	Override:= , 
	BufferMode:= , 
	Options:= , 
	Status=> , 
	Busy=> , 
	Error=> , 
	ErrorID=> );
	

CASE nState OF
	0: //Off
		eState := eBetriebszustand.Off;
		IF bEnable THEN
			nState := 1;
		END_IF
	
	1: //Init
		eState := eBetriebszustand.Init;
		mcPower(Enable := TRUE, Enable_Positive := TRUE,Enable_Negative := TRUE, Axis := ax);
        IF mcPower.Status THEN
            nState := 11;
        END_IF
	
	11: // Homeing
		eState := eBetriebszustand.Init;
		mcHome(
            Execute := TRUE,
            Axis := ax,
            HomingMode := MC_HomingMode.MC_DefaultHoming,
            bCalibrationCam := NOT bSensEndstop
        );
		
		IF mcHome.Done THEN
			bHomeingDone := TRUE;
			mcHome.Execute := FALSE;
			nState := 2;
		END_IF
	
	2: //Ready
		eState := eBetriebszustand.Ready;
		IF bExecute AND bHomeingDone AND NOT bExecuteLast THEN
			nState := 3;
		ELSIF bExecute AND NOT bHomeingDone THEN
			nState := 11;
		END_IF
		bExecuteLast := bExecute;
			
		
	3: //Achsen Bewegung
		eState := eBetriebszustand.Ready;
		IF NOT bMoveing THEN
			mcMoveAbs.Execute := TRUE;
			mcMoveAbs(
				Axis := ax,
				Position := rPosition,
				Velocity := 20.0,
				Acceleration := 50.0,
				Deceleration := 50.0,
				Execute := mcMoveAbs.Execute
			);
			bMoveing := TRUE;
		ELSIF mcMoveAbs.Done THEN
			bMoveing := FALSE;
			nState := 4;
		ELSE
			mcMoveAbs.Execute := FALSE;
			nState := 90;
		END_IF
	
	4: //Done
		eState := eBetriebszustand.Done;
		IF NOT bExecute THEN
			nState := 2;
		END_IF
		
	90: //Error
		eState := eBetriebszustand.Error;
		IF NOT bEnable AND NOT bExecute THEN
			nState := 11;
		END_IF
			
	
		
END_CASE

END_FUNCTION_BLOCK

// ---- POUs/PortalRoboter/FB_Waage_Temp.TcPOU
FUNCTION_BLOCK FB_Waage_Temp
VAR_INPUT
    bEnable  : BOOL;
    bExecute : BOOL;
END_VAR
VAR_OUTPUT
    eState   : eBetriebszustand;
END_VAR
VAR
    timer    : TON;
END_VAR

timer(IN := bEnable AND bExecute, PT := T#1S);

IF bEnable AND bExecute THEN
    eState := eBetriebszustand.Production;

    timer(IN := TRUE);
    IF timer.Q THEN
        eState := eBetriebszustand.Done;
    END_IF
ELSE
    timer(IN := FALSE);
    eState := eBetriebszustand.Ready;
END_IF

END_FUNCTION_BLOCK

// ---- POUs/PortalRoboter/FB_Thermo_Temp.TcPOU
FUNCTION_BLOCK FB_Thermo_Temp
VAR_INPUT
    bEnable  : BOOL;
    bExecute : BOOL;
END_VAR
VAR_OUTPUT
    eState   : eBetriebszustand;
END_VAR
VAR
    timer    : TON;
END_VAR

timer(IN := bEnable AND bExecute, PT := T#2S);

IF bEnable AND bExecute THEN
    eState := eBetriebszustand.Production;

    timer(IN := TRUE);
    IF timer.Q THEN
        eState := eBetriebszustand.Done;
    END_IF
ELSE
    timer(IN := FALSE);
    eState := eBetriebszustand.Ready;
END_IF

END_FUNCTION_BLOCK

// ---- POUs/FB_IotMqttCommunication.TcPOU
FUNCTION_BLOCK FB_IotMqttCommunication
VAR_INPUT
	sTopicToPublish: STRING(255); // MQTT topic
    sMessageToPublish: STRING(255); // Message buffer

END_VAR
VAR_OUTPUT
END_VAR
VAR
	fbMqttClient: FB_IotMqttClient;
	bInitSent : BOOL := FALSE;
	tmrSendMessageInterval: TON := (PT := T#10S); // Interval timer for publishing
END_VAR

fbMqttClient.sHostName := '158.180.44.197';
fbMqttClient.nHostPort := 1883;
fbMqttClient.sTopicPrefix := 'aut/DerGeraet/';
fbMqttClient.sClientId := 'Publishing PLC';
fbMqttClient.sUserName := 'bobm';
fbMqttClient.sUserPassword := 'letmein';
     // MQTT client with initialization
	

fbMqttClient.Execute(bConnect := TRUE);

IF fbMqttClient.bConnected THEN
    tmrSendMessageInterval(IN := TRUE);
	
	IF NOT bInitSent THEN //Init messagees 
		//send Group name
        fbMqttClient.Publish(
            sTopic := '$$groupname',
            pPayload := ADR('DerGreraet'),
            nPayloadSize := LEN('DerGreraet') + 1,
            eQoS := TcIotMqttQos.AtMostOnceDelivery,
            bRetain := TRUE,
            bQueue := FALSE
        );	
		//send group members
        fbMqttClient.Publish(
            sTopic := 'names',
            pPayload := ADR('Naidr, Schulte, Brandt'),
            nPayloadSize := LEN('Naidr, Schulte, Brandt') + 1,
            eQoS := TcIotMqttQos.AtMostOnceDelivery,
            bRetain := TRUE,
            bQueue := FALSE
        );	
		//send unit
        fbMqttClient.Publish(
            sTopic := 'bEnable/$$unit',
            pPayload := ADR('BOOL'),
            nPayloadSize := LEN('BOOL') + 1,
            eQoS := TcIotMqttQos.AtMostOnceDelivery,
            bRetain := TRUE,
            bQueue := FALSE
        );
		bInitSent := TRUE;
	END_IF
	
    IF tmrSendMessageInterval.Q THEN
        tmrSendMessageInterval(IN := FALSE);

        fbMqttClient.Publish(
            sTopic := sTopicToPublish,
            pPayload := ADR(sMessageToPublish),
            nPayloadSize := LEN(sMessageToPublish) + 1,
            eQoS := TcIotMqttQos.AtMostOnceDelivery,
            bRetain := FALSE,
            bQueue := FALSE
        );
    END_IF
END_IF

END_FUNCTION_BLOCK

// ---- POUs/FUN_Scale.TcPOU
FUNCTION FUN_Scale : REAL
VAR_INPUT
	ix : REAL;
	ixmax : REAL;
	ixmin : REAL;
	rymax : REAL;
	rymin : REAL;
END_VAR
VAR
	rk : REAL := 0.085449218;
	rd : REAL := 0;
END_VAR

rk := (rymax - rymin) / (ixmax - ixmin);
rd := rymin - rk * ixmin;

FUN_Scale := rk * ix +rd;

IF FUN_Scale > rymax THEN
	FUN_Scale := rymax;
ELSIF FUN_Scale < rymin THEN
	FUN_Scale := rymin;
END_IF

END_FUNCTION

// ---- POUs/FB_ManipulatorAchsen.TcPOU
FUNCTION_BLOCK FB_ManipulatorAchsen
VAR_INPUT
	bEnable : BOOL;
	bExecute : BOOL;
	rPosition : REAL;
	bRefSens : BOOL;
END_VAR
VAR_OUTPUT
	eState : eBetriebszustand;
END_VAR
VAR
	mcReset : MC_Reset;
	mcPower : MC_Power;
	mcMoveAbsolute : MC_MoveAbsolute;
	mcHome : MC_Home;
	nState : INT;
END_VAR
VAR_IN_OUT
	// Achsen Ref
	ax : Axis_Ref;
END_VAR

END_FUNCTION_BLOCK
